TYPE ST_PiezoStageOL EXTENDS ST_PiezoStage :
STRUCT
    (* Global variables for the TPDO data from the drive. Each one is linked to the respective TPDO channel. *)
    nScantargetPosition	AT %Q*: DINT;
    uScantargetVelocity	AT %Q*: ULINT;
END_STRUCT
END_TYPE

(* stored: Version 1.1.0.1
   DUT ST_PiezoStageOL: Id {f737f5e7-2cd7-4c91-b0fc-92924651ea48} *)
